{attribute 'qualified_only'}
{attribute 'strict'}
{attribute 'to_string'}
TYPE DUT_PathChoice :
(
	Clockwise := 0,
	CounterClockwise := 1
);
END_TYPE

(* stored: Version 1.1.0.1
   EnumerationTextList DUT_PathChoice: Id {a7c9e810-96a5-48b5-a040-34bce75747d7} *)
